// Mitsubishi GX Works2 project: IHW2   PLC: Q03UDE

// global labels: Global1
VAR_GLOBAL
  STARTBUTTON AT X40 : BOOL;
  STOPBUTTON AT X41 : BOOL;
  ESTOPBUTTON AT X42 : BOOL;
  DDXANH1 AT Y50 : BOOL;
  DDVANG1 AT Y51 : BOOL;
  DDDO1 AT Y52 : BOOL;
  DDXANH2 AT Y53 : BOOL;
  DDVANG2 AT Y54 : BOOL;
  DDDO2 AT Y55 : BOOL;
END_VAR

PROGRAM MAIN
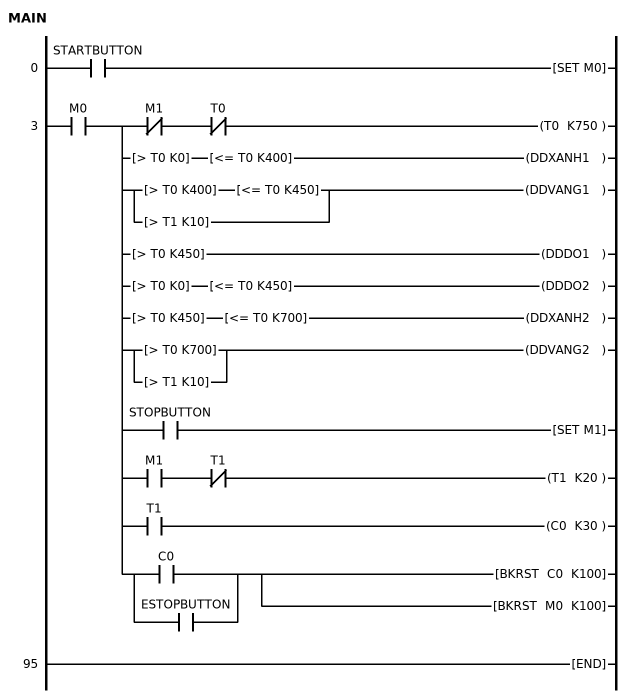
0     LD      STARTBUTTON
      SET     M0
3     LD      M0
      MPS
      ANI     M1
      ANI     T0
      OUT     T0 K750
      MRD
      AND>    T0 K0
      AND<=   T0 K400
      OUT     DDXANH1
      MRD
      LD>     T0 K400
      AND<=   T0 K450
      OR>     T1 K10
      ANB
      OUT     DDVANG1
      MRD
      AND>    T0 K450
      OUT     DDDO1
      MRD
      AND>    T0 K0
      AND<=   T0 K450
      OUT     DDDO2
      MRD
      AND>    T0 K450
      AND<=   T0 K700
      OUT     DDXANH2
      MRD
      LD>     T0 K700
      OR>     T1 K10
      ANB
      OUT     DDVANG2
      MRD
      AND     STOPBUTTON
      SET     M1
      MRD
      AND     M1
      ANI     T1
      OUT     T1 K20
      MRD
      AND     T1
      OUT     C0 K30
      MPP
      LD      C0
      OR      ESTOPBUTTON
      ANB
      BKRST   C0 K100
      BKRST   M0 K100
95    END
END_PROGRAM
